FUNCTION_BLOCK PAEActValve3_3Flange EXTENDS PAEActuator3way
VAR_INPUT
END_VAR
VAR_OUTPUT
END_VAR
VAR
END_VAR

METHOD PUBLIC PAEActValve3_3Flange
VAR_INPUT
END_VAR
END_METHOD

END_FUNCTION_BLOCK

(* stored: Version 1.1.0.1, ProductVersion 3.1.4020.12
   POU PAEActValve3_3Flange: Id {ba3c2330-d4cb-48d1-927f-703d92f22d0f}, SpecialFunc None
   Method PAEActValve3_3Flange: Id {257b0eb3-e992-450f-8644-d75a3599c7fa} *)
